                    IF (Wake_Up < 6000) OR (BMS_Voltage < BMS_Voltage_Min) THEN 
                        (* Transition: '<S1>:358' *)
                        (* Transition: '<S1>:814' *)
                        (* Exit Internal 'POWER_MOTOR_ON': '<S1>:137' *)
                        is_POWER_MOTOR_ON := UPMRacing_14E_StateMachine_IN_NO_ACTIVE_CHILD;
                        is_CAR := UPMRacing_14E_StateMachine_IN_IDLE;
                        (* Entry 'IDLE': '<S1>:333' *)
                        (* '<S1>:333:3' Cooling_Enable = false; *)
                        Cooling_Enable := FALSE;
                        (* '<S1>:333:4' [AMK_TargetVelocity1, AMK_TargetVelocity2, AMK_TargetVelocity3, AMK_TargetVelocity4... *)
                        (* '<S1>:333:5'      ]=Constant(int16(0)); *)
                        (* Simulink Function 'Constant': '<S1>:190' *)
                        x := 0;
                        i0_b_Constant(ssMethodType := SS_OUTPUT, x := x);
                        temp12 := i0_b_Constant.y1;
                        temp13 := i0_b_Constant.y2;
                        temp14 := i0_b_Constant.y3;
                        temp15 := i0_b_Constant.y4;
                        OutportBufferFory4 := temp15;
                        OutportBufferFory3 := temp14;
                        OutportBufferFory2 := temp13;
                        x_l := temp12;
                        AMK_TargetVelocity1 := x_l;
                        AMK_TargetVelocity2 := OutportBufferFory2;
                        AMK_TargetVelocity3 := OutportBufferFory3;
                        AMK_TargetVelocity4 := OutportBufferFory4;
                        (* '<S1>:333:6' [AMK_TorqueLimitPositiv1, AMK_TorqueLimitPositiv2, AMK_TorqueLimitPositiv3,... *)
                        (* '<S1>:333:7'      AMK_TorqueLimitPositiv4]=Constant(int16(0)); *)
                        (* Simulink Function 'Constant': '<S1>:190' *)
                        x := 0;
                        i0_b_Constant(ssMethodType := SS_OUTPUT, x := x);
                        temp12 := i0_b_Constant.y1;
                        temp13 := i0_b_Constant.y2;
                        temp14 := i0_b_Constant.y3;
                        temp15 := i0_b_Constant.y4;
                        OutportBufferFory4 := temp15;
                        OutportBufferFory3 := temp14;
                        OutportBufferFory2 := temp13;
                        x_l := temp12;
                        AMK_TorqueLimitPositiv1 := x_l;
                        AMK_TorqueLimitPositiv2 := OutportBufferFory2;
                        AMK_TorqueLimitPositiv3 := OutportBufferFory3;
                        AMK_TorqueLimitPositiv4 := OutportBufferFory4;
                        (* '<S1>:333:8' [AMK_TorqueLimitNegativ1, AMK_TorqueLimitNegativ2, AMK_TorqueLimitNegativ3, ... *)
                        (* '<S1>:333:9'      AMK_TorqueLimitNegativ4]=Constant(int16(0)); *)
                        (* Simulink Function 'Constant': '<S1>:190' *)
                        x := 0;
                        i0_b_Constant(ssMethodType := SS_OUTPUT, x := x);
                        temp12 := i0_b_Constant.y1;
                        temp13 := i0_b_Constant.y2;
                        temp14 := i0_b_Constant.y3;
                        temp15 := i0_b_Constant.y4;
                        OutportBufferFory4 := temp15;
                        OutportBufferFory3 := temp14;
                        OutportBufferFory2 := temp13;
                        x_l := temp12;
                        AMK_TorqueLimitNegativ1 := x_l;
                        AMK_TorqueLimitNegativ2 := OutportBufferFory2;
                        AMK_TorqueLimitNegativ3 := OutportBufferFory3;
                        AMK_TorqueLimitNegativ4 := OutportBufferFory4;
                        (* Entry Internal 'IDLE': '<S1>:333' *)
                        (* Transition: '<S1>:335' *)
                        is_IDLE := UPMRacing_14E_StateMachine_IN_LVMS_ON;
                        (* Entry 'LVMS_ON': '<S1>:334' *)
                        (* In this state the ECU is waiting to start the inizialization of the inverters *)
                        (* Right now all LV systems are starting to initialize *)
                        (* '<S1>:334:4' Estado = 1; *)
                        Estado := 1;
                        (* Battery relays *)
                        (* '<S1>:334:6' Pre_Charge = false; *)
                        Pre_Charge := FALSE;
                        (* Inverters shutdown *)
                        (* '<S1>:334:8' AMK_bInverterOn1=false; *)
                        AMK_bInverterOn1 := FALSE;
                        (* '<S1>:334:9' AMK_bInverterOn2=false; *)
                        AMK_bInverterOn2 := FALSE;
                        (* '<S1>:334:10' AMK_bInverterOn3=false; *)
                        AMK_bInverterOn3 := FALSE;
                        (* '<S1>:334:11' AMK_bInverterOn4=false; *)
                        AMK_bInverterOn4 := FALSE;
                        (* '<S1>:334:12' AMK_bEnable1=false; *)
                        AMK_bEnable1 := FALSE;
                        (* '<S1>:334:13' AMK_bEnable2=false; *)
                        AMK_bEnable2 := FALSE;
                        (* '<S1>:334:14' AMK_bEnable3=false; *)
                        AMK_bEnable3 := FALSE;
                        (* '<S1>:334:15' AMK_bEnable4=false; *)
                        AMK_bEnable4 := FALSE;
                        (* '<S1>:334:16' AMK_bDcOn1=false; *)
                        AMK_bDcOn1 := FALSE;
                        (* '<S1>:334:17' AMK_bDcOn2=false; *)
                        AMK_bDcOn2 := FALSE;
                        (* '<S1>:334:18' AMK_bDcOn3=false; *)
                        AMK_bDcOn3 := FALSE;
                        (* '<S1>:334:19' AMK_bDcOn4=false; *)
                        AMK_bDcOn4 := FALSE;
                    ELSE 
                        (* '<S1>:814:1' sf_internal_predicateOutput = BMS_Voltage < BMS_Voltage_Min; *)
                        (* Initializes as 0 all control parameters *)
                        (* '<S1>:137:5' [AMK_TargetVelocity1, AMK_TargetVelocity2, AMK_TargetVelocity3, AMK_TargetVelocity4]=Constant(int16(0)) *)
                        (* Simulink Function 'Constant': '<S1>:190' *)
                        x := 0;
                        i0_b_Constant(ssMethodType := SS_OUTPUT, x := x);
                        temp12 := i0_b_Constant.y1;
                        temp13 := i0_b_Constant.y2;
                        temp14 := i0_b_Constant.y3;
                        temp15 := i0_b_Constant.y4;
                        OutportBufferFory4 := temp15;
                        OutportBufferFory3 := temp14;
                        OutportBufferFory2 := temp13;
                        x_l := temp12;
                        AMK_TargetVelocity1 := x_l;
                        AMK_TargetVelocity2 := OutportBufferFory2;
                        AMK_TargetVelocity3 := OutportBufferFory3;
                        AMK_TargetVelocity4 := OutportBufferFory4;
                        (* '<S1>:137:6' [AMK_TorqueLimitPositiv1, AMK_TorqueLimitPositiv2, AMK_TorqueLimitPositiv3, AMK_TorqueLimitPositiv4]=Constant(int16(0)) *)
                        (* Simulink Function 'Constant': '<S1>:190' *)
                        x := 0;
                        i0_b_Constant(ssMethodType := SS_OUTPUT, x := x);
                        temp12 := i0_b_Constant.y1;
                        temp13 := i0_b_Constant.y2;
                        temp14 := i0_b_Constant.y3;
                        temp15 := i0_b_Constant.y4;
                        OutportBufferFory4 := temp15;
                        OutportBufferFory3 := temp14;
                        OutportBufferFory2 := temp13;
                        x_l := temp12;
                        AMK_TorqueLimitPositiv1 := x_l;
                        AMK_TorqueLimitPositiv2 := OutportBufferFory2;
                        AMK_TorqueLimitPositiv3 := OutportBufferFory3;
                        AMK_TorqueLimitPositiv4 := OutportBufferFory4;
                        (* '<S1>:137:7' [AMK_TorqueLimitNegativ1, AMK_TorqueLimitNegativ2, AMK_TorqueLimitNegativ3, AMK_TorqueLimitNegativ4]=Constant(int16(0)) *)
                        (* Simulink Function 'Constant': '<S1>:190' *)
                        x := 0;
                        i0_b_Constant(ssMethodType := SS_OUTPUT, x := x);
                        temp12 := i0_b_Constant.y1;
                        temp13 := i0_b_Constant.y2;
                        temp14 := i0_b_Constant.y3;
                        temp15 := i0_b_Constant.y4;
                        OutportBufferFory4 := temp15;
                        OutportBufferFory3 := temp14;
                        OutportBufferFory2 := temp13;
                        x_l := temp12;
                        AMK_TorqueLimitNegativ1 := x_l;
                        AMK_TorqueLimitNegativ2 := OutportBufferFory2;
                        AMK_TorqueLimitNegativ3 := OutportBufferFory3;
                        AMK_TorqueLimitNegativ4 := OutportBufferFory4;

                        CASE is_POWER_MOTOR_ON OF
                            UPMRacing_14E_StateMachine_IN_HV_STARTUP_1: 
                                (* During 'HV_STARTUP_1': '<S1>:144' *)
                                (* '<S1>:364:1' sf_internal_predicateOutput = AMK_bDcOn1_check==true &amp; AMK_bDcOn2_check==true &amp; AMK_bDcOn3_check==true &amp; AMK_bDcOn4_check==true; *)

                                IF ((AMK_bDcOn1_check AND AMK_bDcOn2_check) AND AMK_bDcOn3_check) AND AMK_bDcOn4_check THEN 
                                    (* Transition: '<S1>:364' *)
                                    is_POWER_MOTOR_ON := UPMRacing_14E_StateMachine_IN_INIT_PRECHARGE;
                                    temporalCounter_i1(timerAction := 1, maxTime := 0);
                                    (* Entry 'INIT_PRECHARGE': '<S1>:440' *)
                                    (* Senal que de inicio a la precarga. En el caso en que volvamos de un error, al detectar directamente *)
                                    (* que se cumple la condicion de salida, no volvera a mandar la senal de iniciar precarga. *)
                                    (* '<S1>:440:4' Estado = 13; *)
                                    Estado := 13;
                                END_IF;

                            UPMRacing_14E_StateMachine_IN_HV_STARTUP_2: 
                                (* During 'HV_STARTUP_2': '<S1>:363' *)
                                (* '<S1>:365:1' sf_internal_predicateOutput = AMK_bEnable1==true &amp; AMK_bEnable2==true &amp; AMK_bEnable3==true &amp; AMK_bEnable4==true; *)

                                IF ((AMK_bEnable1 AND AMK_bEnable2) AND AMK_bEnable3) AND AMK_bEnable4 THEN 
                                    (* Transition: '<S1>:365' *)
                                    is_POWER_MOTOR_ON := UPMRacing_14E_StateMachine_IN_HV_STARTUP_3;
                                    (* Entry 'HV_STARTUP_3': '<S1>:362' *)
                                    (* '<S1>:362:3' AMK_bEnable1=false; *)
                                    AMK_bEnable1 := FALSE;
                                    (* '<S1>:362:4' AMK_bEnable2=false; *)
                                    AMK_bEnable2 := FALSE;
                                    (* '<S1>:362:5' AMK_bEnable3=false; *)
                                    AMK_bEnable3 := FALSE;
                                    (* '<S1>:362:6' AMK_bEnable4=false; *)
                                    AMK_bEnable4 := FALSE;
                                    (* '<S1>:362:7' Estado = 15; *)
                                    Estado := 15;
                                ELSE 
                                    (* Transition: '<S1>:628' *)
                                    (* Transition: '<S1>:627' *)
                                    (* '<S1>:616:1' sf_internal_predicateOutput = Shutdown_Circuit<6000; *)

                                    IF Shutdown_Circuit < 6000 THEN 
                                        (* Transition: '<S1>:616' *)
                                        is_POWER_MOTOR_ON := UPMRacing_14E_StateMachine_IN_NO_ACTIVE_CHILD;
                                        is_CAR := UPMRacing_14E_StateMachine_IN_IDLE;
                                        (* Entry 'IDLE': '<S1>:333' *)
                                        (* '<S1>:333:3' Cooling_Enable = false; *)
                                        Cooling_Enable := FALSE;
                                        (* '<S1>:333:4' [AMK_TargetVelocity1, AMK_TargetVelocity2, AMK_TargetVelocity3, AMK_TargetVelocity4... *)
                                        (* '<S1>:333:5'      ]=Constant(int16(0)); *)
                                        (* Simulink Function 'Constant': '<S1>:190' *)
                                        x := 0;
                                        i0_b_Constant(ssMethodType := SS_OUTPUT, x := x);
                                        temp12 := i0_b_Constant.y1;
                                        temp13 := i0_b_Constant.y2;
                                        temp14 := i0_b_Constant.y3;
                                        temp15 := i0_b_Constant.y4;
                                        OutportBufferFory4 := temp15;
                                        OutportBufferFory3 := temp14;
                                        OutportBufferFory2 := temp13;
                                        x_l := temp12;
                                        AMK_TargetVelocity1 := x_l;
                                        AMK_TargetVelocity2 := OutportBufferFory2;
                                        AMK_TargetVelocity3 := OutportBufferFory3;
                                        AMK_TargetVelocity4 := OutportBufferFory4;
                                        (* '<S1>:333:6' [AMK_TorqueLimitPositiv1, AMK_TorqueLimitPositiv2, AMK_TorqueLimitPositiv3,... *)
                                        (* '<S1>:333:7'      AMK_TorqueLimitPositiv4]=Constant(int16(0)); *)
                                        (* Simulink Function 'Constant': '<S1>:190' *)
                                        x := 0;
                                        i0_b_Constant(ssMethodType := SS_OUTPUT, x := x);
                                        temp12 := i0_b_Constant.y1;
                                        temp13 := i0_b_Constant.y2;
                                        temp14 := i0_b_Constant.y3;
                                        temp15 := i0_b_Constant.y4;
                                        OutportBufferFory4 := temp15;
                                        OutportBufferFory3 := temp14;
                                        OutportBufferFory2 := temp13;
                                        x_l := temp12;
                                        AMK_TorqueLimitPositiv1 := x_l;
                                        AMK_TorqueLimitPositiv2 := OutportBufferFory2;
                                        AMK_TorqueLimitPositiv3 := OutportBufferFory3;
                                        AMK_TorqueLimitPositiv4 := OutportBufferFory4;
                                        (* '<S1>:333:8' [AMK_TorqueLimitNegativ1, AMK_TorqueLimitNegativ2, AMK_TorqueLimitNegativ3, ... *)
                                        (* '<S1>:333:9'      AMK_TorqueLimitNegativ4]=Constant(int16(0)); *)
                                        (* Simulink Function 'Constant': '<S1>:190' *)
                                        x := 0;
                                        i0_b_Constant(ssMethodType := SS_OUTPUT, x := x);
                                        temp12 := i0_b_Constant.y1;
                                        temp13 := i0_b_Constant.y2;
                                        temp14 := i0_b_Constant.y3;
                                        temp15 := i0_b_Constant.y4;
                                        OutportBufferFory4 := temp15;
                                        OutportBufferFory3 := temp14;
                                        OutportBufferFory2 := temp13;
                                        x_l := temp12;
                                        AMK_TorqueLimitNegativ1 := x_l;
                                        AMK_TorqueLimitNegativ2 := OutportBufferFory2;
                                        AMK_TorqueLimitNegativ3 := OutportBufferFory3;
                                        AMK_TorqueLimitNegativ4 := OutportBufferFory4;
                                        is_IDLE := UPMRacing_14E_StateMachine_IN_ERROR_PRECHARGE;
                                        (* Entry 'ERROR_PRECHARGE': '<S1>:617' *)
                                        (* '<S1>:617:2' Estado = 70; *)
                                        Estado := 70;
                                        (* '<S1>:617:3' Pre_Charge = false; *)
                                        Pre_Charge := FALSE;
                                    END_IF;

                                END_IF;

                            UPMRacing_14E_StateMachine_IN_HV_STARTUP_3: 
                                (* During 'HV_STARTUP_3': '<S1>:362' *)
                                (* '<S1>:208:1' sf_internal_predicateOutput = AMK_bEnable1==false &amp; AMK_bEnable2==false &amp; AMK_bEnable3==false &amp; AMK_bEnable4==false; *)

                                IF ((( NOT AMK_bEnable1) AND ( NOT AMK_bEnable2)) AND ( NOT AMK_bEnable3)) AND ( NOT AMK_bEnable4) THEN 
                                    (* Transition: '<S1>:208' *)
                                    is_POWER_MOTOR_ON := UPMRacing_14E_StateMachine_IN_HV_STARTUP_4;
                                    (* Entry 'HV_STARTUP_4': '<S1>:139' *)
                                    (* '<S1>:139:3' AMK_bEnable1=true; *)
                                    AMK_bEnable1 := TRUE;
                                    (* '<S1>:139:4' AMK_bEnable2=true; *)
                                    AMK_bEnable2 := TRUE;
                                    (* '<S1>:139:5' AMK_bEnable3=true; *)
                                    AMK_bEnable3 := TRUE;
                                    (* '<S1>:139:6' AMK_bEnable4=true; *)
                                    AMK_bEnable4 := TRUE;
                                    (* '<S1>:139:7' Estado = 16; *)
                                    Estado := 16;
                                ELSE 
                                    (* Transition: '<S1>:629' *)
                                    (* Transition: '<S1>:626' *)
                                    (* Transition: '<S1>:627' *)
                                    (* '<S1>:616:1' sf_internal_predicateOutput = Shutdown_Circuit<6000; *)

                                    IF Shutdown_Circuit < 6000 THEN 
                                        (* Transition: '<S1>:616' *)
                                        is_POWER_MOTOR_ON := UPMRacing_14E_StateMachine_IN_NO_ACTIVE_CHILD;
                                        is_CAR := UPMRacing_14E_StateMachine_IN_IDLE;
                                        (* Entry 'IDLE': '<S1>:333' *)
                                        (* '<S1>:333:3' Cooling_Enable = false; *)
                                        Cooling_Enable := FALSE;
                                        (* '<S1>:333:4' [AMK_TargetVelocity1, AMK_TargetVelocity2, AMK_TargetVelocity3, AMK_TargetVelocity4... *)
                                        (* '<S1>:333:5'      ]=Constant(int16(0)); *)
                                        (* Simulink Function 'Constant': '<S1>:190' *)
                                        x := 0;
                                        i0_b_Constant(ssMethodType := SS_OUTPUT, x := x);
                                        temp12 := i0_b_Constant.y1;
                                        temp13 := i0_b_Constant.y2;
                                        temp14 := i0_b_Constant.y3;
                                        temp15 := i0_b_Constant.y4;
                                        OutportBufferFory4 := temp15;
                                        OutportBufferFory3 := temp14;
                                        OutportBufferFory2 := temp13;
                                        x_l := temp12;
                                        AMK_TargetVelocity1 := x_l;
                                        AMK_TargetVelocity2 := OutportBufferFory2;
                                        AMK_TargetVelocity3 := OutportBufferFory3;
                                        AMK_TargetVelocity4 := OutportBufferFory4;
                                        (* '<S1>:333:6' [AMK_TorqueLimitPositiv1, AMK_TorqueLimitPositiv2, AMK_TorqueLimitPositiv3,... *)
                                        (* '<S1>:333:7'      AMK_TorqueLimitPositiv4]=Constant(int16(0)); *)
                                        (* Simulink Function 'Constant': '<S1>:190' *)
                                        x := 0;
                                        i0_b_Constant(ssMethodType := SS_OUTPUT, x := x);
                                        temp12 := i0_b_Constant.y1;
                                        temp13 := i0_b_Constant.y2;
                                        temp14 := i0_b_Constant.y3;
                                        temp15 := i0_b_Constant.y4;
                                        OutportBufferFory4 := temp15;
                                        OutportBufferFory3 := temp14;
                                        OutportBufferFory2 := temp13;
                                        x_l := temp12;
                                        AMK_TorqueLimitPositiv1 := x_l;
                                        AMK_TorqueLimitPositiv2 := OutportBufferFory2;
                                        AMK_TorqueLimitPositiv3 := OutportBufferFory3;
                                        AMK_TorqueLimitPositiv4 := OutportBufferFory4;
                                        (* '<S1>:333:8' [AMK_TorqueLimitNegativ1, AMK_TorqueLimitNegativ2, AMK_TorqueLimitNegativ3, ... *)
                                        (* '<S1>:333:9'      AMK_TorqueLimitNegativ4]=Constant(int16(0)); *)
                                        (* Simulink Function 'Constant': '<S1>:190' *)
                                        x := 0;
                                        i0_b_Constant(ssMethodType := SS_OUTPUT, x := x);
                                        temp12 := i0_b_Constant.y1;
                                        temp13 := i0_b_Constant.y2;
                                        temp14 := i0_b_Constant.y3;
                                        temp15 := i0_b_Constant.y4;
                                        OutportBufferFory4 := temp15;
                                        OutportBufferFory3 := temp14;
                                        OutportBufferFory2 := temp13;
                                        x_l := temp12;
                                        AMK_TorqueLimitNegativ1 := x_l;
                                        AMK_TorqueLimitNegativ2 := OutportBufferFory2;
                                        AMK_TorqueLimitNegativ3 := OutportBufferFory3;
                                        AMK_TorqueLimitNegativ4 := OutportBufferFory4;
                                        is_IDLE := UPMRacing_14E_StateMachine_IN_ERROR_PRECHARGE;
                                        (* Entry 'ERROR_PRECHARGE': '<S1>:617' *)
                                        (* '<S1>:617:2' Estado = 70; *)
                                        Estado := 70;
                                        (* '<S1>:617:3' Pre_Charge = false; *)
                                        Pre_Charge := FALSE;
                                    END_IF;

                                END_IF;

                            UPMRacing_14E_StateMachine_IN_HV_STARTUP_4: 
                                (* During 'HV_STARTUP_4': '<S1>:139' *)
                                (* '<S1>:367:1' sf_internal_predicateOutput = AMK_bEnable1==true &amp;  AMK_bEnable2==true &amp; ... *)
                                (* '<S1>:367:2'  AMK_bEnable3==true &amp; AMK_bEnable4==true; *)

                                IF ((AMK_bEnable1 AND AMK_bEnable2) AND AMK_bEnable3) AND AMK_bEnable4 THEN 
                                    (* Transition: '<S1>:367' *)
                                    is_POWER_MOTOR_ON := UPMRacing_14E_StateMachine_IN_HV_STARTUP_5;
                                    (* Entry 'HV_STARTUP_5': '<S1>:366' *)
                                    (* '<S1>:366:3' AMK_bInverterOn1=true; *)
                                    AMK_bInverterOn1 := TRUE;
                                    (* '<S1>:366:4' AMK_bInverterOn2=true; *)
                                    AMK_bInverterOn2 := TRUE;
                                    (* '<S1>:366:5' AMK_bInverterOn3=true; *)
                                    AMK_bInverterOn3 := TRUE;
                                    (* '<S1>:366:6' AMK_bInverterOn4=true; *)
                                    AMK_bInverterOn4 := TRUE;
                                    (* '<S1>:366:7' Estado = 17; *)
                                    Estado := 17;
                                ELSE 
                                    (* Transition: '<S1>:630' *)
                                    (* Transition: '<S1>:625' *)
                                    (* Transition: '<S1>:626' *)
                                    (* Transition: '<S1>:627' *)
                                    (* '<S1>:616:1' sf_internal_predicateOutput = Shutdown_Circuit<6000; *)

                                    IF Shutdown_Circuit < 6000 THEN 
                                        (* Transition: '<S1>:616' *)
                                        is_POWER_MOTOR_ON := UPMRacing_14E_StateMachine_IN_NO_ACTIVE_CHILD;
                                        is_CAR := UPMRacing_14E_StateMachine_IN_IDLE;
                                        (* Entry 'IDLE': '<S1>:333' *)
                                        (* '<S1>:333:3' Cooling_Enable = false; *)
                                        Cooling_Enable := FALSE;
                                        (* '<S1>:333:4' [AMK_TargetVelocity1, AMK_TargetVelocity2, AMK_TargetVelocity3, AMK_TargetVelocity4... *)
                                        (* '<S1>:333:5'      ]=Constant(int16(0)); *)
                                        (* Simulink Function 'Constant': '<S1>:190' *)
                                        x := 0;
                                        i0_b_Constant(ssMethodType := SS_OUTPUT, x := x);
                                        temp12 := i0_b_Constant.y1;
                                        temp13 := i0_b_Constant.y2;
                                        temp14 := i0_b_Constant.y3;
                                        temp15 := i0_b_Constant.y4;
                                        OutportBufferFory4 := temp15;
                                        OutportBufferFory3 := temp14;
                                        OutportBufferFory2 := temp13;
                                        x_l := temp12;
                                        AMK_TargetVelocity1 := x_l;
                                        AMK_TargetVelocity2 := OutportBufferFory2;
                                        AMK_TargetVelocity3 := OutportBufferFory3;
                                        AMK_TargetVelocity4 := OutportBufferFory4;
                                        (* '<S1>:333:6' [AMK_TorqueLimitPositiv1, AMK_TorqueLimitPositiv2, AMK_TorqueLimitPositiv3,... *)
                                        (* '<S1>:333:7'      AMK_TorqueLimitPositiv4]=Constant(int16(0)); *)
                                        (* Simulink Function 'Constant': '<S1>:190' *)
                                        x := 0;
                                        i0_b_Constant(ssMethodType := SS_OUTPUT, x := x);
                                        temp12 := i0_b_Constant.y1;
                                        temp13 := i0_b_Constant.y2;
                                        temp14 := i0_b_Constant.y3;
                                        temp15 := i0_b_Constant.y4;
                                        OutportBufferFory4 := temp15;
                                        OutportBufferFory3 := temp14;
                                        OutportBufferFory2 := temp13;
                                        x_l := temp12;
                                        AMK_TorqueLimitPositiv1 := x_l;
                                        AMK_TorqueLimitPositiv2 := OutportBufferFory2;
                                        AMK_TorqueLimitPositiv3 := OutportBufferFory3;
                                        AMK_TorqueLimitPositiv4 := OutportBufferFory4;
                                        (* '<S1>:333:8' [AMK_TorqueLimitNegativ1, AMK_TorqueLimitNegativ2, AMK_TorqueLimitNegativ3, ... *)
                                        (* '<S1>:333:9'      AMK_TorqueLimitNegativ4]=Constant(int16(0)); *)
                                        (* Simulink Function 'Constant': '<S1>:190' *)
                                        x := 0;
                                        i0_b_Constant(ssMethodType := SS_OUTPUT, x := x);
                                        temp12 := i0_b_Constant.y1;
                                        temp13 := i0_b_Constant.y2;
                                        temp14 := i0_b_Constant.y3;
                                        temp15 := i0_b_Constant.y4;
                                        OutportBufferFory4 := temp15;
                                        OutportBufferFory3 := temp14;
                                        OutportBufferFory2 := temp13;
                                        x_l := temp12;
                                        AMK_TorqueLimitNegativ1 := x_l;
                                        AMK_TorqueLimitNegativ2 := OutportBufferFory2;
                                        AMK_TorqueLimitNegativ3 := OutportBufferFory3;
                                        AMK_TorqueLimitNegativ4 := OutportBufferFory4;
                                        is_IDLE := UPMRacing_14E_StateMachine_IN_ERROR_PRECHARGE;
                                        (* Entry 'ERROR_PRECHARGE': '<S1>:617' *)
                                        (* '<S1>:617:2' Estado = 70; *)
                                        Estado := 70;
                                        (* '<S1>:617:3' Pre_Charge = false; *)
                                        Pre_Charge := FALSE;
                                    END_IF;

                                END_IF;

                            UPMRacing_14E_StateMachine_IN_HV_STARTUP_5: 
                                (* During 'HV_STARTUP_5': '<S1>:366' *)
                                (* '<S1>:262:1' sf_internal_predicateOutput = AMK_bInverterOn1_check==true &amp;  AMK_bInverterOn2_check==true &amp; ... *)
                                (* '<S1>:262:2'  AMK_bInverterOn3_check==true &amp; AMK_bInverterOn4_check==true; *)

                                IF ((AMK_bInverterOn1_check AND AMK_bInverterOn2_check) AND AMK_bInverterOn3_check) AND AMK_bInverterOn4_check THEN 
                                    (* Transition: '<S1>:262' *)
                                    is_POWER_MOTOR_ON := UPMRacing_14E_StateMachine_IN_HV_STARTUP_6;
                                    (* Entry 'HV_STARTUP_6': '<S1>:259' *)
                                    (* AMK_X140_BE2_INV_1=true; *)
                                    (* AMK_X140_BE2_INV_2=true; *)
                                    (* AMK_X140_BE2_INV_3=true; *)
                                    (* AMK_X140_BE2_INV_4=true; *)
                                    (* '<S1>:259:7' Estado = 18; *)
                                    Estado := 18;
                                ELSE 
                                    (* Transition: '<S1>:631' *)
                                    (* Transition: '<S1>:624' *)
                                    (* Transition: '<S1>:625' *)
                                    (* Transition: '<S1>:626' *)
                                    (* Transition: '<S1>:627' *)
                                    (* '<S1>:616:1' sf_internal_predicateOutput = Shutdown_Circuit<6000; *)

                                    IF Shutdown_Circuit < 6000 THEN 
                                        (* Transition: '<S1>:616' *)
                                        is_POWER_MOTOR_ON := UPMRacing_14E_StateMachine_IN_NO_ACTIVE_CHILD;
                                        is_CAR := UPMRacing_14E_StateMachine_IN_IDLE;
                                        (* Entry 'IDLE': '<S1>:333' *)
                                        (* '<S1>:333:3' Cooling_Enable = false; *)
                                        Cooling_Enable := FALSE;
                                        (* '<S1>:333:4' [AMK_TargetVelocity1, AMK_TargetVelocity2, AMK_TargetVelocity3, AMK_TargetVelocity4... *)
                                        (* '<S1>:333:5'      ]=Constant(int16(0)); *)
                                        (* Simulink Function 'Constant': '<S1>:190' *)
                                        x := 0;
                                        i0_b_Constant(ssMethodType := SS_OUTPUT, x := x);
                                        temp12 := i0_b_Constant.y1;
                                        temp13 := i0_b_Constant.y2;
                                        temp14 := i0_b_Constant.y3;
                                        temp15 := i0_b_Constant.y4;
                                        OutportBufferFory4 := temp15;
                                        OutportBufferFory3 := temp14;
                                        OutportBufferFory2 := temp13;
                                        x_l := temp12;
                                        AMK_TargetVelocity1 := x_l;
                                        AMK_TargetVelocity2 := OutportBufferFory2;
                                        AMK_TargetVelocity3 := OutportBufferFory3;
                                        AMK_TargetVelocity4 := OutportBufferFory4;
                                        (* '<S1>:333:6' [AMK_TorqueLimitPositiv1, AMK_TorqueLimitPositiv2, AMK_TorqueLimitPositiv3,... *)
                                        (* '<S1>:333:7'      AMK_TorqueLimitPositiv4]=Constant(int16(0)); *)
                                        (* Simulink Function 'Constant': '<S1>:190' *)
                                        x := 0;
                                        i0_b_Constant(ssMethodType := SS_OUTPUT, x := x);
                                        temp12 := i0_b_Constant.y1;
                                        temp13 := i0_b_Constant.y2;
                                        temp14 := i0_b_Constant.y3;
                                        temp15 := i0_b_Constant.y4;
                                        OutportBufferFory4 := temp15;
                                        OutportBufferFory3 := temp14;
                                        OutportBufferFory2 := temp13;
                                        x_l := temp12;
                                        AMK_TorqueLimitPositiv1 := x_l;
                                        AMK_TorqueLimitPositiv2 := OutportBufferFory2;
                                        AMK_TorqueLimitPositiv3 := OutportBufferFory3;
                                        AMK_TorqueLimitPositiv4 := OutportBufferFory4;
                                        (* '<S1>:333:8' [AMK_TorqueLimitNegativ1, AMK_TorqueLimitNegativ2, AMK_TorqueLimitNegativ3, ... *)
                                        (* '<S1>:333:9'      AMK_TorqueLimitNegativ4]=Constant(int16(0)); *)
                                        (* Simulink Function 'Constant': '<S1>:190' *)
                                        x := 0;
                                        i0_b_Constant(ssMethodType := SS_OUTPUT, x := x);
                                        temp12 := i0_b_Constant.y1;
                                        temp13 := i0_b_Constant.y2;
                                        temp14 := i0_b_Constant.y3;
                                        temp15 := i0_b_Constant.y4;
                                        OutportBufferFory4 := temp15;
                                        OutportBufferFory3 := temp14;
                                        OutportBufferFory2 := temp13;
                                        x_l := temp12;
                                        AMK_TorqueLimitNegativ1 := x_l;
                                        AMK_TorqueLimitNegativ2 := OutportBufferFory2;
                                        AMK_TorqueLimitNegativ3 := OutportBufferFory3;
                                        AMK_TorqueLimitNegativ4 := OutportBufferFory4;
                                        is_IDLE := UPMRacing_14E_StateMachine_IN_ERROR_PRECHARGE;
                                        (* Entry 'ERROR_PRECHARGE': '<S1>:617' *)
                                        (* '<S1>:617:2' Estado = 70; *)
                                        Estado := 70;
                                        (* '<S1>:617:3' Pre_Charge = false; *)
                                        Pre_Charge := FALSE;
                                    END_IF;

                                END_IF;

                            UPMRacing_14E_StateMachine_IN_HV_STARTUP_6: 
                                (* During 'HV_STARTUP_6': '<S1>:259' *)
                                (* '<S1>:147:1' sf_internal_predicateOutput = AMK_bQuitInverterOn1==true &amp;  AMK_bQuitInverterOn2==true... *)
                                (* '<S1>:147:2'  &amp; AMK_bQuitInverterOn3==true &amp; AMK_bQuitInverterOn4==true... *)
                                (* '<S1>:147:3' &amp; Drive_Button < 12000; *)

                                IF (((AMK_bQuitInverterOn1 AND AMK_bQuitInverterOn2) AND AMK_bQuitInverterOn3) AND AMK_bQuitInverterOn4) AND (Drive_Button < 12000) THEN 
                                    (* Transition: '<S1>:147' *)
                                    is_POWER_MOTOR_ON := UPMRacing_14E_StateMachine_IN_NO_ACTIVE_CHILD;
                                    is_CAR := UPMRacing_14E_StateMachine_IN_DRIVE;
                                    (* Entry 'DRIVE': '<S1>:169' *)
                                    (* '<S1>:169:2' Cooling_Enable = true; *)
                                    Cooling_Enable := TRUE;
                                    (* Entry Internal 'DRIVE': '<S1>:169' *)
                                    (* Transition: '<S1>:264' *)
                                    is_DRIVE := UPMRacing_14E_StateMachine_IN_PRE_DRIVE;
                                    (* Entry 'PRE_DRIVE': '<S1>:503' *)
                                    (* '<S1>:503:2' Estado = 20; *)
                                    Estado := 20;
                                ELSE 
                                    (* Transition: '<S1>:634' *)
                                    (* Transition: '<S1>:633' *)
                                    (* Transition: '<S1>:624' *)
                                    (* Transition: '<S1>:625' *)
                                    (* Transition: '<S1>:626' *)
                                    (* Transition: '<S1>:627' *)
                                    (* '<S1>:616:1' sf_internal_predicateOutput = Shutdown_Circuit<6000; *)

                                    IF Shutdown_Circuit < 6000 THEN 
                                        (* Transition: '<S1>:616' *)
                                        is_POWER_MOTOR_ON := UPMRacing_14E_StateMachine_IN_NO_ACTIVE_CHILD;
                                        is_CAR := UPMRacing_14E_StateMachine_IN_IDLE;
                                        (* Entry 'IDLE': '<S1>:333' *)
                                        (* '<S1>:333:3' Cooling_Enable = false; *)
                                        Cooling_Enable := FALSE;
                                        (* '<S1>:333:4' [AMK_TargetVelocity1, AMK_TargetVelocity2, AMK_TargetVelocity3, AMK_TargetVelocity4... *)
                                        (* '<S1>:333:5'      ]=Constant(int16(0)); *)
                                        (* Simulink Function 'Constant': '<S1>:190' *)
                                        x := 0;
                                        i0_b_Constant(ssMethodType := SS_OUTPUT, x := x);
                                        temp12 := i0_b_Constant.y1;
                                        temp13 := i0_b_Constant.y2;
                                        temp14 := i0_b_Constant.y3;
                                        temp15 := i0_b_Constant.y4;
                                        OutportBufferFory4 := temp15;
                                        OutportBufferFory3 := temp14;
                                        OutportBufferFory2 := temp13;
                                        x_l := temp12;
                                        AMK_TargetVelocity1 := x_l;
                                        AMK_TargetVelocity2 := OutportBufferFory2;
                                        AMK_TargetVelocity3 := OutportBufferFory3;
                                        AMK_TargetVelocity4 := OutportBufferFory4;
                                        (* '<S1>:333:6' [AMK_TorqueLimitPositiv1, AMK_TorqueLimitPositiv2, AMK_TorqueLimitPositiv3,... *)
                                        (* '<S1>:333:7'      AMK_TorqueLimitPositiv4]=Constant(int16(0)); *)
                                        (* Simulink Function 'Constant': '<S1>:190' *)
                                        x := 0;
                                        i0_b_Constant(ssMethodType := SS_OUTPUT, x := x);
                                        temp12 := i0_b_Constant.y1;
                                        temp13 := i0_b_Constant.y2;
                                        temp14 := i0_b_Constant.y3;
                                        temp15 := i0_b_Constant.y4;
                                        OutportBufferFory4 := temp15;
                                        OutportBufferFory3 := temp14;
                                        OutportBufferFory2 := temp13;
                                        x_l := temp12;
                                        AMK_TorqueLimitPositiv1 := x_l;
                                        AMK_TorqueLimitPositiv2 := OutportBufferFory2;
                                        AMK_TorqueLimitPositiv3 := OutportBufferFory3;
                                        AMK_TorqueLimitPositiv4 := OutportBufferFory4;
                                        (* '<S1>:333:8' [AMK_TorqueLimitNegativ1, AMK_TorqueLimitNegativ2, AMK_TorqueLimitNegativ3, ... *)
                                        (* '<S1>:333:9'      AMK_TorqueLimitNegativ4]=Constant(int16(0)); *)
                                        (* Simulink Function 'Constant': '<S1>:190' *)
                                        x := 0;
                                        i0_b_Constant(ssMethodType := SS_OUTPUT, x := x);
                                        temp12 := i0_b_Constant.y1;
                                        temp13 := i0_b_Constant.y2;
                                        temp14 := i0_b_Constant.y3;
                                        temp15 := i0_b_Constant.y4;
                                        OutportBufferFory4 := temp15;
                                        OutportBufferFory3 := temp14;
                                        OutportBufferFory2 := temp13;
                                        x_l := temp12;
                                        AMK_TorqueLimitNegativ1 := x_l;
                                        AMK_TorqueLimitNegativ2 := OutportBufferFory2;
                                        AMK_TorqueLimitNegativ3 := OutportBufferFory3;
                                        AMK_TorqueLimitNegativ4 := OutportBufferFory4;
                                        is_IDLE := UPMRacing_14E_StateMachine_IN_ERROR_PRECHARGE;
                                        (* Entry 'ERROR_PRECHARGE': '<S1>:617' *)
                                        (* '<S1>:617:2' Estado = 70; *)
                                        Estado := 70;
                                        (* '<S1>:617:3' Pre_Charge = false; *)
                                        Pre_Charge := FALSE;
                                    END_IF;

                                END_IF;

                            UPMRacing_14E_StateMachine_IN_INIT_PRECHARGE: 
                                (* During 'INIT_PRECHARGE': '<S1>:440' *)
                                (* '<S1>:441:1' sf_internal_predicateOutput = AMK_bQuitDcOn1==true &amp; AMK_bQuitDcOn2==true &amp; AMK_bQuitDcOn3==true &amp; AMK_bQuitDcOn4==true; *)

                                IF ((AMK_bQuitDcOn1 AND AMK_bQuitDcOn2) AND AMK_bQuitDcOn3) AND AMK_bQuitDcOn4 THEN 
                                    (* Transition: '<S1>:441' *)
                                    is_POWER_MOTOR_ON := UPMRacing_14E_StateMachine_IN_HV_STARTUP_2;
                                    (* Entry 'HV_STARTUP_2': '<S1>:363' *)
                                    (* '<S1>:363:3' AMK_bEnable1=true; *)
                                    AMK_bEnable1 := TRUE;
                                    (* '<S1>:363:4' AMK_bEnable2=true; *)
                                    AMK_bEnable2 := TRUE;
                                    (* '<S1>:363:5' AMK_bEnable3=true; *)
                                    AMK_bEnable3 := TRUE;
                                    (* '<S1>:363:6' AMK_bEnable4=true; *)
                                    AMK_bEnable4 := TRUE;
                                    (* '<S1>:363:7' Estado = 14; *)
                                    Estado := 14;
                                ELSE 
                                    (* '<S1>:615:1' sf_internal_predicateOutput = after(2,sec); *)
                                    temporalCounter_i1(timerAction := 2, maxTime := 2000);

                                    IF temporalCounter_i1.done THEN 
                                        (* Transition: '<S1>:615' *)
                                        (* '<S1>:616:1' sf_internal_predicateOutput = Shutdown_Circuit<6000; *)

                                        IF Shutdown_Circuit < 6000 THEN 
                                            (* Transition: '<S1>:616' *)
                                            is_POWER_MOTOR_ON := UPMRacing_14E_StateMachine_IN_NO_ACTIVE_CHILD;
                                            is_CAR := UPMRacing_14E_StateMachine_IN_IDLE;
                                            (* Entry 'IDLE': '<S1>:333' *)
                                            (* '<S1>:333:3' Cooling_Enable = false; *)
                                            Cooling_Enable := FALSE;
                                            (* '<S1>:333:4' [AMK_TargetVelocity1, AMK_TargetVelocity2, AMK_TargetVelocity3, AMK_TargetVelocity4... *)
                                            (* '<S1>:333:5'      ]=Constant(int16(0)); *)
                                            (* Simulink Function 'Constant': '<S1>:190' *)
                                            x := 0;
                                            i0_b_Constant(ssMethodType := SS_OUTPUT, x := x);
                                            temp12 := i0_b_Constant.y1;
                                            temp13 := i0_b_Constant.y2;
                                            temp14 := i0_b_Constant.y3;
                                            temp15 := i0_b_Constant.y4;
                                            OutportBufferFory4 := temp15;
                                            OutportBufferFory3 := temp14;
                                            OutportBufferFory2 := temp13;
                                            x_l := temp12;
                                            AMK_TargetVelocity1 := x_l;
                                            AMK_TargetVelocity2 := OutportBufferFory2;
                                            AMK_TargetVelocity3 := OutportBufferFory3;
                                            AMK_TargetVelocity4 := OutportBufferFory4;
                                            (* '<S1>:333:6' [AMK_TorqueLimitPositiv1, AMK_TorqueLimitPositiv2, AMK_TorqueLimitPositiv3,... *)
                                            (* '<S1>:333:7'      AMK_TorqueLimitPositiv4]=Constant(int16(0)); *)
                                            (* Simulink Function 'Constant': '<S1>:190' *)
                                            x := 0;
                                            i0_b_Constant(ssMethodType := SS_OUTPUT, x := x);
                                            temp12 := i0_b_Constant.y1;
                                            temp13 := i0_b_Constant.y2;
                                            temp14 := i0_b_Constant.y3;
                                            temp15 := i0_b_Constant.y4;
                                            OutportBufferFory4 := temp15;
                                            OutportBufferFory3 := temp14;
                                            OutportBufferFory2 := temp13;
                                            x_l := temp12;
                                            AMK_TorqueLimitPositiv1 := x_l;
                                            AMK_TorqueLimitPositiv2 := OutportBufferFory2;
                                            AMK_TorqueLimitPositiv3 := OutportBufferFory3;
                                            AMK_TorqueLimitPositiv4 := OutportBufferFory4;
                                            (* '<S1>:333:8' [AMK_TorqueLimitNegativ1, AMK_TorqueLimitNegativ2, AMK_TorqueLimitNegativ3, ... *)
                                            (* '<S1>:333:9'      AMK_TorqueLimitNegativ4]=Constant(int16(0)); *)
                                            (* Simulink Function 'Constant': '<S1>:190' *)
                                            x := 0;
                                            i0_b_Constant(ssMethodType := SS_OUTPUT, x := x);
                                            temp12 := i0_b_Constant.y1;
                                            temp13 := i0_b_Constant.y2;
                                            temp14 := i0_b_Constant.y3;
                                            temp15 := i0_b_Constant.y4;
                                            OutportBufferFory4 := temp15;
                                            OutportBufferFory3 := temp14;
                                            OutportBufferFory2 := temp13;
                                            x_l := temp12;
                                            AMK_TorqueLimitNegativ1 := x_l;
                                            AMK_TorqueLimitNegativ2 := OutportBufferFory2;
                                            AMK_TorqueLimitNegativ3 := OutportBufferFory3;
                                            AMK_TorqueLimitNegativ4 := OutportBufferFory4;
                                            is_IDLE := UPMRacing_14E_StateMachine_IN_ERROR_PRECHARGE;
                                            (* Entry 'ERROR_PRECHARGE': '<S1>:617' *)
                                            (* '<S1>:617:2' Estado = 70; *)
                                            Estado := 70;
                                            (* '<S1>:617:3' Pre_Charge = false; *)
                                            Pre_Charge := FALSE;
                                        ELSE 
                                            (* Senal que de inicio a la precarga. En el caso en que volvamos de un error, al detectar directamente *)
                                            (* que se cumple la condicion de salida, no volvera a mandar la senal de iniciar precarga. *)
                                            (* '<S1>:440:6' Pre_Charge=true; *)
                                            Pre_Charge := TRUE;
                                        END_IF;

                                    ELSE 
                                        (* Senal que de inicio a la precarga. En el caso en que volvamos de un error, al detectar directamente *)
                                        (* que se cumple la condicion de salida, no volvera a mandar la senal de iniciar precarga. *)
                                        (* '<S1>:440:6' Pre_Charge=true; *)
                                        Pre_Charge := TRUE;
                                    END_IF;

                                END_IF;

                            ELSE
                                (* During 'INVERTER_ON': '<S1>:163' *)
                                (* '<S1>:164:1' sf_internal_predicateOutput = AMK_bSystemReady1==true &amp; AMK_bSystemReady2==true &amp; AMK_bSystemReady3==true &amp;... *)
                                (* '<S1>:164:2' AMK_bSystemReady4==true; *)

                                IF ((AMK_bSystemReady1 AND AMK_bSystemReady2) AND AMK_bSystemReady3) AND AMK_bSystemReady4 THEN 
                                    (* Transition: '<S1>:164' *)
                                    is_POWER_MOTOR_ON := UPMRacing_14E_StateMachine_IN_HV_STARTUP_1;
                                    (* Entry 'HV_STARTUP_1': '<S1>:144' *)
                                    (* '<S1>:144:3' AMK_bDcOn1=true; *)
                                    AMK_bDcOn1 := TRUE;
                                    (* '<S1>:144:4' AMK_bDcOn2=true; *)
                                    AMK_bDcOn2 := TRUE;
                                    (* '<S1>:144:5' AMK_bDcOn3=true; *)
                                    AMK_bDcOn3 := TRUE;
                                    (* '<S1>:144:6' AMK_bDcOn4=true; *)
                                    AMK_bDcOn4 := TRUE;
                                    (* '<S1>:144:7' Estado = 12; *)
                                    Estado := 12;
                                END_IF;

                        END_CASE;

                    END_IF;

                ELSE
                    (* During 'SHUTDOWN_SEQUENCE': '<S1>:189' *)

                    CASE is_SHUTDOWN_SEQUENCE OF
                        UPMRacing_14E_StateMachine_IN_HV_SHUTDOWN: 
                            (* During 'HV_SHUTDOWN': '<S1>:216' *)
                            (* '<S1>:473:1' sf_internal_predicateOutput = AMK_bDcOn1_check==false &amp; AMK_bDcOn2_check==false &amp; AMK_bDcOn3_check==false &amp; AMK_bDcOn4_check==false; *)

                            IF ((( NOT AMK_bDcOn1_check) AND ( NOT AMK_bDcOn2_check)) AND ( NOT AMK_bDcOn3_check)) AND ( NOT AMK_bDcOn4_check) THEN 
                                (* Transition: '<S1>:473' *)
                                is_SHUTDOWN_SEQUENCE := UPMRacing_14E_StateMachine_IN_INIT_DISCHARGE;
                                temporalCounter_i1(timerAction := 1, maxTime := 0);
                                (* Entry 'INIT_DISCHARGE': '<S1>:472' *)
                                (* '<S1>:472:2' Estado = 33; *)
                                Estado := 33;
                            ELSE 
                                (* '<S1>:216:2' Estado = 32; *)
                                Estado := 32;
                                (* AMK_X140_BE1_INV_1=false; *)
                                (* AMK_X140_BE1_INV_2=false; *)
                                (* AMK_X140_BE1_INV_3=false; *)
                                (* AMK_X140_BE1_INV_4=false; *)
                                (* '<S1>:216:7' AMK_bDcOn1=false; *)
                                AMK_bDcOn1 := FALSE;
                                (* '<S1>:216:8' AMK_bDcOn2=false; *)
                                AMK_bDcOn2 := FALSE;
                                (* '<S1>:216:9' AMK_bDcOn3=false; *)
                                AMK_bDcOn3 := FALSE;
                                (* '<S1>:216:10' AMK_bDcOn4=false; *)
                                AMK_bDcOn4 := FALSE;
                            END_IF;

                        UPMRacing_14E_StateMachine_IN_INIT_DISCHARGE: 
                            (* During 'INIT_DISCHARGE': '<S1>:472' *)
                            (* '<S1>:476:1' sf_internal_predicateOutput = (Pre_Charge == false) &amp; (Shutdown_Circuit < 6000); *)

                            IF ( NOT Pre_Charge) AND (Shutdown_Circuit < 6000) THEN 
                                (* Transition: '<S1>:476' *)
                                (* '<S1>:477:1' sf_internal_predicateOutput = after(5,sec); *)
                                temporalCounter_i1(timerAction := 2, maxTime := 5000);

                                IF temporalCounter_i1.done THEN 
                                    (* Transition: '<S1>:477' *)
                                    is_SHUTDOWN_SEQUENCE := UPMRacing_14E_StateMachine_IN_INIT_DISCHARGE1;
                                    (* Entry 'INIT_DISCHARGE1': '<S1>:474' *)
                                    (* '<S1>:474:2' Estado = 34; *)
                                    Estado := 34;
                                END_IF;

                            ELSE 
                                (* '<S1>:472:4' Pre_Charge = false; *)
                                Pre_Charge := FALSE;
                            END_IF;

                        UPMRacing_14E_StateMachine_IN_INIT_DISCHARGE1: 
                            (* During 'INIT_DISCHARGE1': '<S1>:474' *)
                            (* '<S1>:221:1' sf_internal_predicateOutput = AMK_bQuitDcOn1==false &amp; AMK_bQuitDcOn2==false &amp;  AMK_bQuitDcOn3==false &amp; AMK_bQuitDcOn1==false &amp; Wake_Up < 6000; *)
                            sf_internal_predicateOutput :=  NOT AMK_bQuitDcOn1;

                            IF (((sf_internal_predicateOutput AND ( NOT AMK_bQuitDcOn2)) AND ( NOT AMK_bQuitDcOn3)) AND sf_internal_predicateOutput) AND (Wake_Up < 6000) THEN 
                                (* Transition: '<S1>:221' *)
                                is_SHUTDOWN_SEQUENCE := UPMRacing_14E_StateMachine_IN_NO_ACTIVE_CHILD;
                                is_CAR := UPMRacing_14E_StateMachine_IN_IDLE;
                                (* Entry 'IDLE': '<S1>:333' *)
                                (* '<S1>:333:3' Cooling_Enable = false; *)
                                Cooling_Enable := FALSE;
                                (* '<S1>:333:4' [AMK_TargetVelocity1, AMK_TargetVelocity2, AMK_TargetVelocity3, AMK_TargetVelocity4... *)
                                (* '<S1>:333:5'      ]=Constant(int16(0)); *)
                                (* Simulink Function 'Constant': '<S1>:190' *)
                                x := 0;
                                i0_b_Constant(ssMethodType := SS_OUTPUT, x := x);
                                temp12 := i0_b_Constant.y1;
                                temp13 := i0_b_Constant.y2;
                                temp14 := i0_b_Constant.y3;
                                temp15 := i0_b_Constant.y4;
                                OutportBufferFory4 := temp15;
                                OutportBufferFory3 := temp14;
                                OutportBufferFory2 := temp13;
                                x_l := temp12;
                                AMK_TargetVelocity1 := x_l;
                                AMK_TargetVelocity2 := OutportBufferFory2;
                                AMK_TargetVelocity3 := OutportBufferFory3;
                                AMK_TargetVelocity4 := OutportBufferFory4;
                                (* '<S1>:333:6' [AMK_TorqueLimitPositiv1, AMK_TorqueLimitPositiv2, AMK_TorqueLimitPositiv3,... *)
                                (* '<S1>:333:7'      AMK_TorqueLimitPositiv4]=Constant(int16(0)); *)
                                (* Simulink Function 'Constant': '<S1>:190' *)
                                x := 0;
                                i0_b_Constant(ssMethodType := SS_OUTPUT, x := x);
                                temp12 := i0_b_Constant.y1;
                                temp13 := i0_b_Constant.y2;
                                temp14 := i0_b_Constant.y3;
                                temp15 := i0_b_Constant.y4;
                                OutportBufferFory4 := temp15;
                                OutportBufferFory3 := temp14;
                                OutportBufferFory2 := temp13;
                                x_l := temp12;
                                AMK_TorqueLimitPositiv1 := x_l;
                                AMK_TorqueLimitPositiv2 := OutportBufferFory2;
                                AMK_TorqueLimitPositiv3 := OutportBufferFory3;
                                AMK_TorqueLimitPositiv4 := OutportBufferFory4;
                                (* '<S1>:333:8' [AMK_TorqueLimitNegativ1, AMK_TorqueLimitNegativ2, AMK_TorqueLimitNegativ3, ... *)
                                (* '<S1>:333:9'      AMK_TorqueLimitNegativ4]=Constant(int16(0)); *)
                                (* Simulink Function 'Constant': '<S1>:190' *)
                                x := 0;
                                i0_b_Constant(ssMethodType := SS_OUTPUT, x := x);
                                temp12 := i0_b_Constant.y1;
                                temp13 := i0_b_Constant.y2;
                                temp14 := i0_b_Constant.y3;
                                temp15 := i0_b_Constant.y4;
                                OutportBufferFory4 := temp15;
                                OutportBufferFory3 := temp14;
                                OutportBufferFory2 := temp13;
                                x_l := temp12;
                                AMK_TorqueLimitNegativ1 := x_l;
                                AMK_TorqueLimitNegativ2 := OutportBufferFory2;
                                AMK_TorqueLimitNegativ3 := OutportBufferFory3;
                                AMK_TorqueLimitNegativ4 := OutportBufferFory4;
                                (* Entry Internal 'IDLE': '<S1>:333' *)
                                (* Transition: '<S1>:335' *)
                                is_IDLE := UPMRacing_14E_StateMachine_IN_LVMS_ON;
                                (* Entry 'LVMS_ON': '<S1>:334' *)
                                (* In this state the ECU is waiting to start the inizialization of the inverters *)
                                (* Right now all LV systems are starting to initialize *)
                                (* '<S1>:334:4' Estado = 1; *)
                                Estado := 1;
                                (* Battery relays *)
                                (* '<S1>:334:6' Pre_Charge = false; *)
                                Pre_Charge := FALSE;
                                (* Inverters shutdown *)
                                (* '<S1>:334:8' AMK_bInverterOn1=false; *)
                                AMK_bInverterOn1 := FALSE;
                                (* '<S1>:334:9' AMK_bInverterOn2=false; *)
                                AMK_bInverterOn2 := FALSE;
                                (* '<S1>:334:10' AMK_bInverterOn3=false; *)
                                AMK_bInverterOn3 := FALSE;
                                (* '<S1>:334:11' AMK_bInverterOn4=false; *)
                                AMK_bInverterOn4 := FALSE;
                                (* '<S1>:334:12' AMK_bEnable1=false; *)
                                AMK_bEnable1 := FALSE;
                                (* '<S1>:334:13' AMK_bEnable2=false; *)
                                AMK_bEnable2 := FALSE;
                                (* '<S1>:334:14' AMK_bEnable3=false; *)
                                AMK_bEnable3 := FALSE;
                                (* '<S1>:334:15' AMK_bEnable4=false; *)
                                AMK_bEnable4 := FALSE;
                                (* '<S1>:334:16' AMK_bDcOn1=false; *)
                                AMK_bDcOn1 := FALSE;
                                (* '<S1>:334:17' AMK_bDcOn2=false; *)
                                AMK_bDcOn2 := FALSE;
                                (* '<S1>:334:18' AMK_bDcOn3=false; *)
                                AMK_bDcOn3 := FALSE;
                                (* '<S1>:334:19' AMK_bDcOn4=false; *)
                                AMK_bDcOn4 := FALSE;
                            END_IF;

                        ELSE
                            (* During 'INVERTER_CONTROLLER_SHUTDOWN': '<S1>:212' *)
                            (* '<S1>:217:1' sf_internal_predicateOutput = AMK_bQuitInverterOn1==false &amp; AMK_bQuitInverterOn2==false &amp;  AMK_bQuitInverterOn3==false &amp; AMK_bQuitInverterOn4==false... *)
                            (* '<S1>:217:2' &amp; AMK_bInverterOn1_check==false &amp;  AMK_bInverterOn2_check==false &amp;  AMK_bInverterOn3_check==false &amp; AMK_bInverterOn4_check==false; *)

                            IF ((((((( NOT AMK_bQuitInverterOn1) AND ( NOT AMK_bQuitInverterOn2)) AND ( NOT AMK_bQuitInverterOn3)) AND ( NOT AMK_bQuitInverterOn4)) AND ( NOT AMK_bInverterOn1_check)) AND ( NOT AMK_bInverterOn2_check)) AND ( NOT AMK_bInverterOn3_check)) AND ( NOT AMK_bInverterOn4_check) THEN 
                                (* Transition: '<S1>:217' *)
                                is_SHUTDOWN_SEQUENCE := UPMRacing_14E_StateMachine_IN_HV_SHUTDOWN;
                                (* Entry 'HV_SHUTDOWN': '<S1>:216' *)
                            ELSE 
                                (* '<S1>:212:2' Estado = 31; *)
                                Estado := 31;
                                (* AMK_X140_BE2_INV_1=false; *)
                                (* AMK_X140_BE2_INV_2=false; *)
                                (* AMK_X140_BE2_INV_3=false; *)
                                (* AMK_X140_BE2_INV_4=false; *)
                                (* '<S1>:212:7' AMK_bInverterOn1=false; *)
                                AMK_bInverterOn1 := FALSE;
                                (* '<S1>:212:8' AMK_bInverterOn2=false; *)
                                AMK_bInverterOn2 := FALSE;
                                (* '<S1>:212:9' AMK_bInverterOn3=false; *)
                                AMK_bInverterOn3 := FALSE;
                                (* '<S1>:212:10' AMK_bInverterOn4=false; *)
                                AMK_bInverterOn4 := FALSE;
                                (* '<S1>:212:11' AMK_bEnable1=false; *)
                                AMK_bEnable1 := FALSE;
                                (* '<S1>:212:12' AMK_bEnable2=false; *)
                                AMK_bEnable2 := FALSE;
                                (* '<S1>:212:13' AMK_bEnable3=false; *)
                                AMK_bEnable3 := FALSE;
                                (* '<S1>:212:14' AMK_bEnable4=false; *)
                                AMK_bEnable4 := FALSE;
                            END_IF;

                    END_CASE;

            END_CASE;


            IF temp9 THEN 
                (* Exit Internal 'DRIVE': '<S1>:169' *)

                CASE is_DRIVE OF
                    UPMRacing_14E_StateMachine_IN_RTDS: 
                        (* Exit 'RTDS': '<S1>:555' *)
                        (* '<S1>:555:8' RTDS_Sound = false; *)
                        RTDS_Sound := FALSE;
                        is_DRIVE := UPMRacing_14E_StateMachine_IN_NO_ACTIVE_CHILD;
                    ELSE
                        is_DRIVE := UPMRacing_14E_StateMachine_IN_NO_ACTIVE_CHILD;
                END_CASE;

                is_CAR := UPMRacing_14E_StateMachine_IN_SHUTDOWN_SEQUENCE;
                (* Entry 'SHUTDOWN_SEQUENCE': '<S1>:189' *)
                (* '<S1>:189:3' [AMK_TorqueLimitNegativ1,AMK_TorqueLimitNegativ2,AMK_TorqueLimitNegativ3,AMK_TorqueLimitNegativ4]=Constant(int16(0)); *)
                (* Simulink Function 'Constant': '<S1>:190' *)
                x := 0;
                i0_b_Constant(ssMethodType := SS_OUTPUT, x := x);
                temp12 := i0_b_Constant.y1;
                temp13 := i0_b_Constant.y2;
                temp14 := i0_b_Constant.y3;
                temp15 := i0_b_Constant.y4;
                OutportBufferFory4 := temp15;
                OutportBufferFory3 := temp14;
                OutportBufferFory2 := temp13;
                x_l := temp12;
                AMK_TorqueLimitNegativ1 := x_l;
                AMK_TorqueLimitNegativ2 := OutportBufferFory2;
                AMK_TorqueLimitNegativ3 := OutportBufferFory3;
                AMK_TorqueLimitNegativ4 := OutportBufferFory4;
                (* '<S1>:189:4' [AMK_TargetVelocity1, AMK_TargetVelocity2, AMK_TargetVelocity3,AMK_TargetVelocity4]=Constant(int16(0)); *)
                (* Simulink Function 'Constant': '<S1>:190' *)
                x := 0;
                i0_b_Constant(ssMethodType := SS_OUTPUT, x := x);
                temp12 := i0_b_Constant.y1;
                temp13 := i0_b_Constant.y2;
                temp14 := i0_b_Constant.y3;
                temp15 := i0_b_Constant.y4;
                OutportBufferFory4 := temp15;
                OutportBufferFory3 := temp14;
                OutportBufferFory2 := temp13;
                x_l := temp12;
                AMK_TargetVelocity1 := x_l;
                AMK_TargetVelocity2 := OutportBufferFory2;
                AMK_TargetVelocity3 := OutportBufferFory3;
                AMK_TargetVelocity4 := OutportBufferFory4;
                (* '<S1>:189:5' [AMK_TorqueLimitPositiv1, AMK_TorqueLimitPositiv2, AMK_TorqueLimitPositiv3,AMK_TorqueLimitPositiv4]=Constant(int16(0)); *)
                (* Simulink Function 'Constant': '<S1>:190' *)
                x := 0;
                i0_b_Constant(ssMethodType := SS_OUTPUT, x := x);
                temp12 := i0_b_Constant.y1;
                temp13 := i0_b_Constant.y2;
                temp14 := i0_b_Constant.y3;
                temp15 := i0_b_Constant.y4;
                OutportBufferFory4 := temp15;
                OutportBufferFory3 := temp14;
                OutportBufferFory2 := temp13;
                x_l := temp12;
                AMK_TorqueLimitPositiv1 := x_l;
                AMK_TorqueLimitPositiv2 := OutportBufferFory2;
                AMK_TorqueLimitPositiv3 := OutportBufferFory3;
                AMK_TorqueLimitPositiv4 := OutportBufferFory4;
                (* '<S1>:189:6' Cooling_Enable = true; *)
                Cooling_Enable := TRUE;
                (* Entry Internal 'SHUTDOWN_SEQUENCE': '<S1>:189' *)
                (* Transition: '<S1>:345' *)
                is_SHUTDOWN_SEQUENCE := UPMRacing_14E_StateMachine_IN_INVERTER_CONTROLLER_SHUTDOWN;
                (* Entry 'INVERTER_CONTROLLER_SHUTDOWN': '<S1>:212' *)
            END_IF;


            IF temp8 THEN 
                is_DRIVE := UPMRacing_14E_StateMachine_IN_BRAKE;
                (* Entry 'BRAKE': '<S1>:170' *)
                (* '<S1>:170:2' Estado = 22; *)
                Estado := 22;
            END_IF;


            IF temp10 THEN 
                is_DRIVE := UPMRacing_14E_StateMachine_IN_Accelerate;
                (* Entry 'Accelerate': '<S1>:146' *)
                (* '<S1>:146:2' Estado = 21; *)
                Estado := 21;
            END_IF;

            (* During 'ERROR_INVERTER': '<S1>:381' *)
            (* '<S1>:381:2' [Inverter_Error,Inverter_Warning] = Error_Control(AMK_bError1,AMK_bError2,AMK_bError3,AMK_bError4,AMK_bWarn1,AMK_bWarn2,AMK_bWarn3,AMK_bWarn4); *)
            (* Simulink Function 'Error_Control': '<S1>:390' *)
            b_AMK_bError1 := AMK_bError1;
            b_AMK_bError2 := AMK_bError2;
            b_AMK_bError3 := AMK_bError3;
            b_AMK_bError4 := AMK_bError4;
            b_AMK_bWarn1 := AMK_bWarn1;
            b_AMK_bWarn2 := AMK_bWarn2;
            b_AMK_bWarn3 := AMK_bWarn3;
            b_AMK_bWarn4 := AMK_bWarn4;
            i0_Error_Control(ssMethodType := SS_OUTPUT, AMK_bError1 := b_AMK_bError1, AMK_bError2 := b_AMK_bError2, AMK_bError3 := b_AMK_bError3, AMK_bError4 := b_AMK_bError4, AMK_bWarn1 := b_AMK_bWarn1, AMK_bWarn2 := b_AMK_bWarn2, AMK_bWarn3 := b_AMK_bWarn3, AMK_bWarn4 := b_AMK_bWarn4);
            sf_internal_predicateOutput := i0_Error_Control.Inverter_Error;
            temp10 := i0_Error_Control.Inverter_Warning;
            LogicalOperator1 := temp10;
            LogicalOperator := sf_internal_predicateOutput;
            Inverter_Error := LogicalOperator;
            Inverter_Warning := LogicalOperator1;

            CASE is_ERROR_INVERTER OF
                UPMRacing_14E_StateMachine_IN_ERROR: 
                    (* Outport: '<Root>/Estado_Error' *)
                    Estado_Error := 12;
                    (* During 'ERROR': '<S1>:385' *)
                    (* '<S1>:388:1' sf_internal_predicateOutput = Inverter_Error == 0; *)

                    IF  NOT LogicalOperator THEN 
                        (* Transition: '<S1>:388' *)
                        is_ERROR_INVERTER := UPMRacing_14E_StateMachine_IN_NO_ERROR;
                        (* Outport: '<Root>/Estado_Error' *)
                        (* Entry 'NO_ERROR': '<S1>:384' *)
                        (* No hay errores *)
                        (* '<S1>:384:3' Estado_Error = 11; *)
                        Estado_Error := 11;
                    ELSE 
                        (* '<S1>:435:1' sf_internal_predicateOutput = Reset_Button > 3000; *)

                        IF Reset_Button > 3000 THEN 
                            (* Transition: '<S1>:435' *)
                            is_ERROR_INVERTER := UPMRacing_14E_StateMachine_IN_RESET_ERROR;
                            (* Outport: '<Root>/Estado_Error' *)
                            (* Entry 'RESET_ERROR': '<S1>:403' *)
                            (* Reseteamos errores *)
                            (* '<S1>:403:3' Estado_Error = 13; *)
                            Estado_Error := 13;
                        ELSE 
                            (* Hay errores *)
                            (* Esperar a boton de reset para resetear errores *)
                            (* '<S1>:385:6' Info_Inverter_Error = Error_Info(AMK_ErrorInfo1,AMK_ErrorInfo2,AMK_ErrorInfo3,AMK_ErrorInfo4,... *)
                            (* '<S1>:385:7'     AMK_bError1,AMK_bError2,AMK_bError3,AMK_bError4) *)
                            (* Simulink Function 'Error_Info': '<S1>:463' *)
                            b_AMK_ErrorInfo1 := AMK_ErrorInfo1;
                            b_AMK_ErrorInfo2 := AMK_ErrorInfo2;
                            b_AMK_ErrorInfo3 := AMK_ErrorInfo3;
                            b_AMK_ErrorInfo4 := AMK_ErrorInfo4;
                            AMK_bError1_b := AMK_bError1;
                            AMK_bError2_h := AMK_bError2;
                            AMK_bError3_d := AMK_bError3;
                            AMK_bError4_a := AMK_bError4;
                            i0_Error_Info(ssMethodType := SS_OUTPUT, AMK_ErrorInfo1 := b_AMK_ErrorInfo1, AMK_ErrorInfo2 := b_AMK_ErrorInfo2, AMK_ErrorInfo3 := b_AMK_ErrorInfo3, AMK_ErrorInfo4 := b_AMK_ErrorInfo4, AMK_bError1 := AMK_bError1_b, AMK_bError2 := AMK_bError2_h, AMK_bError3 := AMK_bError3_d, AMK_bError4 := AMK_bError4_a);
                            temp7 := i0_Error_Info.Info_Inverter_Error;
                            b_Add := temp7;
                            Info_Inverter_Error := b_Add;
                        END_IF;

                    END_IF;

                UPMRacing_14E_StateMachine_IN_NO_ERROR: 
                    (* Outport: '<Root>/Estado_Error' *)
                    Estado_Error := 11;
                    (* During 'NO_ERROR': '<S1>:384' *)
                    (* '<S1>:386:1' sf_internal_predicateOutput = Inverter_Error==1 &amp; Reset_Button == 0; *)

                    IF LogicalOperator AND (Reset_Button = 0) THEN 
                        (* Transition: '<S1>:386' *)
                        is_ERROR_INVERTER := UPMRacing_14E_StateMachine_IN_ERROR;
                        (* Outport: '<Root>/Estado_Error' *)
                        (* Entry 'ERROR': '<S1>:385' *)
                        (* Hay errores *)
                        (* Esperar a boton de reset para resetear errores *)
                        (* '<S1>:385:4' Estado_Error = 12; *)
                        Estado_Error := 12;
                    END_IF;

                ELSE
                    (* Outport: '<Root>/Estado_Error' *)
                    Estado_Error := 13;
                    (* During 'RESET_ERROR': '<S1>:403' *)
                    (* '<S1>:436:1' sf_internal_predicateOutput = Reset_Button < 300; *)

                    IF Reset_Button < 300 THEN 
                        (* Transition: '<S1>:436' *)
                        (* Exit 'RESET_ERROR': '<S1>:403' *)
                        (* '<S1>:403:6' Info_Inverter_Error = 0; *)
                        Info_Inverter_Error := 0;
                        is_ERROR_INVERTER := UPMRacing_14E_StateMachine_IN_NO_ERROR;
                        (* Outport: '<Root>/Estado_Error' incorporates:
                         *  Outport: '<Root>/Info_Inverter_Error' *)
                        (* Entry 'NO_ERROR': '<S1>:384' *)
                        (* No hay errores *)
                        (* '<S1>:384:3' Estado_Error = 11; *)
                        Estado_Error := 11;
                    ELSE 
                        (* Reseteamos errores *)
                        (* '<S1>:403:5' [AMK_bErrorReset1,AMK_bErrorReset2,AMK_bErrorReset3,AMK_bErrorReset4] = Error_RESET *)
                        (* Simulink Function 'Error_RESET': '<S1>:414' *)
                        i0_Error_RESET(ssMethodType := SS_OUTPUT);
                        sf_internal_predicateOutput := i0_Error_RESET.AMK_bErrorReset1;
                        temp10 := i0_Error_RESET.AMK_bErrorReset2;
                        temp8 := i0_Error_RESET.AMK_bErrorReset3;
                        temp9 := i0_Error_RESET.AMK_bErrorReset4;
                        OutportBufferForAMK_bErrorReset4 := temp9;
                        OutportBufferForAMK_bErrorReset3 := temp8;
                        OutportBufferForAMK_bErrorReset2 := temp10;
                        Compare := sf_internal_predicateOutput;
                        AMK_bErrorReset1 := Compare;
                        AMK_bErrorReset2 := OutportBufferForAMK_bErrorReset2;
                        AMK_bErrorReset3 := OutportBufferForAMK_bErrorReset3;
                        AMK_bErrorReset4 := OutportBufferForAMK_bErrorReset4;
                    END_IF;

            END_CASE;

            (* During 'BRAKE_LIGHT': '<S1>:519' *)

            CASE is_BRAKE_LIGHT OF
                UPMRacing_14E_StateMachine_IN_LIGHT_OFF: 
                    (* During 'LIGHT_OFF': '<S1>:520' *)
                    (* '<S1>:523:1' sf_internal_predicateOutput = Brake_Pedal <= Braking_OffSet; *)

                    IF Brake_Pedal <= Braking_OffSet THEN 
                        (* Transition: '<S1>:523' *)
                        is_BRAKE_LIGHT := UPMRacing_14E_StateMachine_IN_LIGHT_ON;
                        (* Entry 'LIGHT_ON': '<S1>:522' *)
                    ELSE 
                        (* '<S1>:520:3' Brake_Light = false; *)
                        Brake_Light := FALSE;
                    END_IF;

                ELSE
                    (* During 'LIGHT_ON': '<S1>:522' *)
                    (* '<S1>:524:1' sf_internal_predicateOutput = Brake_Pedal > Braking_OffSet; *)

                    IF Brake_Pedal > Braking_OffSet THEN 
                        (* Transition: '<S1>:524' *)
                        is_BRAKE_LIGHT := UPMRacing_14E_StateMachine_IN_LIGHT_OFF;
                        (* Entry 'LIGHT_OFF': '<S1>:520' *)
                    ELSE 
                        (* '<S1>:522:3' Brake_Light = true; *)
                        Brake_Light := TRUE;
                    END_IF;

            END_CASE;

            (* During 'COOLING_RIGHT': '<S1>:526' *)

            CASE is_COOLING_RIGHT OF
                UPMRacing_14E_StateMachine_IN_COOLING_OFF_RIGHT: 
                    (* During 'COOLING_OFF_RIGHT': '<S1>:612' *)
                    (* '<S1>:611:1' sf_internal_predicateOutput = Cooling_Enable == true; *)

                    IF Cooling_Enable THEN 
                        (* Transition: '<S1>:611' *)
                        (* Exit 'COOLING_OFF_RIGHT': '<S1>:612' *)
                        (* '<S1>:612:4' Cooling_Pumps_On = false; *)
                        Cooling_Pumps_On := FALSE;
                        is_COOLING_RIGHT := UPMRacing_14E_StateMachine_IN_FAN_OFF;
                        (* Entry 'FAN_OFF': '<S1>:527' *)
                    END_IF;

                UPMRacing_14E_StateMachine_IN_FAN_OFF: 
                    (* During 'FAN_OFF': '<S1>:527' *)
                    (* '<S1>:531:1' sf_internal_predicateOutput = (AMK_TempMotor1 > Motor_Upper_Temp) || ... *)
                    (* '<S1>:531:2' (AMK_TempMotor3 > Motor_Upper_Temp); *)

                    IF (AMK_TempMotor1 > Motor_Upper_Temp) OR (AMK_TempMotor3 > Motor_Upper_Temp) THEN 
                        (* Transition: '<S1>:531' *)
                        is_COOLING_RIGHT := UPMRacing_14E_StateMachine_IN_FAN_ON;
                        (* Entry 'FAN_ON': '<S1>:530' *)
                    ELSE 
                        (* '<S1>:609:1' sf_internal_predicateOutput = Cooling_Enable == false; *)

                        IF  NOT Cooling_Enable THEN 
                            (* Transition: '<S1>:609' *)
                            is_COOLING_RIGHT := UPMRacing_14E_StateMachine_IN_COOLING_OFF_RIGHT;
                            (* Entry 'COOLING_OFF_RIGHT': '<S1>:612' *)
                            (* '<S1>:612:2' Cooling_Pumps_On = false; *)
                            Cooling_Pumps_On := FALSE;
                            (* '<S1>:612:3' Fan_Left = false; *)
                            Fan_Left := FALSE;
                        ELSE 
                            (* '<S1>:527:2' Fan_Right = false; *)
                            Fan_Right := FALSE;
                        END_IF;

                    END_IF;

                UPMRacing_14E_StateMachine_IN_FAN_OFF_Speed: 
                    (* During 'FAN_OFF_Speed': '<S1>:533' *)
                    (* '<S1>:534:1' sf_internal_predicateOutput = Speed<Fan_Lower_Speed; *)

                    IF Speed < UINT_TO_REAL(Fan_Lower_Speed) THEN 
                        (* Transition: '<S1>:534' *)
                        is_COOLING_RIGHT := UPMRacing_14E_StateMachine_IN_FAN_ON;
                        (* Entry 'FAN_ON': '<S1>:530' *)
                    ELSE 
                        (* '<S1>:607:1' sf_internal_predicateOutput = Cooling_Enable == false; *)

                        IF  NOT Cooling_Enable THEN 
                            (* Transition: '<S1>:607' *)
                            is_COOLING_RIGHT := UPMRacing_14E_StateMachine_IN_COOLING_OFF_RIGHT;
                            (* Entry 'COOLING_OFF_RIGHT': '<S1>:612' *)
                            (* '<S1>:612:2' Cooling_Pumps_On = false; *)
                            Cooling_Pumps_On := FALSE;
                            (* '<S1>:612:3' Fan_Left = false; *)
                            Fan_Left := FALSE;
                        ELSE 
                            (* '<S1>:533:2' Fan_Right = false; *)
                            Fan_Right := FALSE;
                        END_IF;

                    END_IF;

                ELSE
                    (* During 'FAN_ON': '<S1>:530' *)
                    (* '<S1>:532:1' sf_internal_predicateOutput = (AMK_TempMotor1 < Motor_Lower_Temp) || ... *)
                    (* '<S1>:532:2' (AMK_TempMotor3 < Motor_Lower_Temp); *)

                    IF (AMK_TempMotor1 < Motor_Lower_Temp) OR (AMK_TempMotor3 < Motor_Lower_Temp) THEN 
                        (* Transition: '<S1>:532' *)
                        is_COOLING_RIGHT := UPMRacing_14E_StateMachine_IN_FAN_OFF;
                        (* Entry 'FAN_OFF': '<S1>:527' *)
                    ELSE 
                        (* '<S1>:608:1' sf_internal_predicateOutput = Cooling_Enable == false; *)

                        IF  NOT Cooling_Enable THEN 
                            (* Transition: '<S1>:608' *)
                            is_COOLING_RIGHT := UPMRacing_14E_StateMachine_IN_COOLING_OFF_RIGHT;
                            (* Entry 'COOLING_OFF_RIGHT': '<S1>:612' *)
                            (* '<S1>:612:2' Cooling_Pumps_On = false; *)
                            Cooling_Pumps_On := FALSE;
                            (* '<S1>:612:3' Fan_Left = false; *)
                            Fan_Left := FALSE;
                        ELSE 
                            (* '<S1>:535:1' sf_internal_predicateOutput = Speed>Fan_Upper_Speed; *)

                            IF Speed > UINT_TO_REAL(Fan_Upper_Speed) THEN 
                                (* Transition: '<S1>:535' *)
                                is_COOLING_RIGHT := UPMRacing_14E_StateMachine_IN_FAN_OFF_Speed;
                                (* Entry 'FAN_OFF_Speed': '<S1>:533' *)
                            ELSE 
                                (* '<S1>:530:2' Fan_Right = false; *)
                                Fan_Right := FALSE;
                            END_IF;

                        END_IF;

                    END_IF;

            END_CASE;

            (* During 'COOLING_LEFT': '<S1>:543' *)
            (* '<S1>:543:3' [AIM_TempInverter1,AIM_TempInverter2,AIM_TempInverter3,AIM_TempInverter4] = Temp_Inverter(AMK_TempInverter1,AMK_TempInverter2,AMK_TempInverter3,AMK_TempInverter4); *)
            (* Simulink Function 'Temp_Inverter': '<S1>:577' *)
            b_AMK_TempInverter1 := AMK_TempInverter1;
            b_AMK_TempInverter2 := AMK_TempInverter2;
            b_AMK_TempInverter3 := AMK_TempInverter3;
            b_AMK_TempInverter4 := AMK_TempInverter4;
            i0_Temp_Inverter(ssMethodType := SS_OUTPUT, AMK_TempInverter1 := b_AMK_TempInverter1, AMK_TempInverter2 := b_AMK_TempInverter2, AMK_TempInverter3 := b_AMK_TempInverter3, AMK_TempInverter4 := b_AMK_TempInverter4);
            temp3 := i0_Temp_Inverter.AIM_TempInverter1;
            temp4 := i0_Temp_Inverter.AIM_TempInverter2;
            temp5 := i0_Temp_Inverter.AIM_TempInverter3;
            temp6 := i0_Temp_Inverter.AIM_TempInverter4;
            DataTypeConversion3_e := temp6;
            DataTypeConversion1_c := temp5;
            DataTypeConversion2_f := temp4;
            DataTypeConversion_h := temp3;
            AIM_TempInverter1 := DataTypeConversion_h;
            AIM_TempInverter2 := DataTypeConversion2_f;
            AIM_TempInverter3 := DataTypeConversion1_c;
            AIM_TempInverter4 := DataTypeConversion3_e;
            (* '<S1>:543:4' [AIM_TempMotor1,AIM_TempMotor2,AIM_TempMotor3,AIM_TempMotor4] = Temp_Motor(AMK_TempMotor1,AMK_TempMotor2,AMK_TempMotor3,AMK_TempMotor4); *)
            (* Simulink Function 'Temp_Motor': '<S1>:593' *)
            b_AMK_TempMotor1 := AMK_TempMotor1;
            b_AMK_TempMotor2 := AMK_TempMotor2;
            b_AMK_TempMotor3 := AMK_TempMotor3;
            b_AMK_TempMotor4 := AMK_TempMotor4;
            i0_Temp_Motor(ssMethodType := SS_OUTPUT, AMK_TempMotor1 := b_AMK_TempMotor1, AMK_TempMotor2 := b_AMK_TempMotor2, AMK_TempMotor3 := b_AMK_TempMotor3, AMK_TempMotor4 := b_AMK_TempMotor4);
            temp3 := i0_Temp_Motor.AIM_TempMotor1;
            temp4 := i0_Temp_Motor.AIM_TempMotor2;
            temp5 := i0_Temp_Motor.AIM_TempMotor3;
            temp6 := i0_Temp_Motor.AIM_TempMotor4;
            DataTypeConversion3_p := temp6;
            DataTypeConversion1_g := temp5;
            DataTypeConversion2_e := temp4;
            DataTypeConversion_e := temp3;
            AIM_TempMotor1 := DataTypeConversion_e;
            AIM_TempMotor2 := DataTypeConversion2_e;
            AIM_TempMotor3 := DataTypeConversion1_g;
            AIM_TempMotor4 := DataTypeConversion3_p;
            (* '<S1>:543:5' [AIM_TempIGBT1,AIM_TempIGBT2,AIM_TempIGBT3,AIM_TempIGBT4] = Temp_IGBT(AMK_TempIGBT1,AMK_TempIGBT2,AMK_TempIGBT3,AMK_TempIGBT4); *)
            (* Simulink Function 'Temp_IGBT': '<S1>:644' *)
            b_AMK_TempIGBT1 := AMK_TempIGBT1;
            b_AMK_TempIGBT2 := AMK_TempIGBT2;
            b_AMK_TempIGBT3 := AMK_TempIGBT3;
            b_AMK_TempIGBT4 := AMK_TempIGBT4;
            i0_Temp_IGBT(ssMethodType := SS_OUTPUT, AMK_TempIGBT1 := b_AMK_TempIGBT1, AMK_TempIGBT2 := b_AMK_TempIGBT2, AMK_TempIGBT3 := b_AMK_TempIGBT3, AMK_TempIGBT4 := b_AMK_TempIGBT4);
            temp3 := i0_Temp_IGBT.AIM_TempIGBT1;
            temp4 := i0_Temp_IGBT.AIM_TempIGBT2;
            temp5 := i0_Temp_IGBT.AIM_TempIGBT3;
            temp6 := i0_Temp_IGBT.AIM_TempIGBT4;
            DataTypeConversion3_o := temp6;
            DataTypeConversion1_n := temp5;
            DataTypeConversion2_m := temp4;
            DataTypeConversion_b := temp3;
            AIM_TempIGBT1 := DataTypeConversion_b;
            AIM_TempIGBT2 := DataTypeConversion2_m;
            AIM_TempIGBT3 := DataTypeConversion1_n;
            AIM_TempIGBT4 := DataTypeConversion3_o;
            (* '<S1>:543:6' [AIM_bDerating1,AIM_bDerating2,AIM_bDerating3,AIM_bDerating4] = Derating(AMK_bDerating1,AMK_bDerating2,AMK_bDerating3,AMK_bDerating4); *)
            (* Simulink Function 'Derating': '<S1>:711' *)
            b_AMK_bDerating1 := AMK_bDerating1;
            b_AMK_bDerating2 := AMK_bDerating2;
            b_AMK_bDerating3 := AMK_bDerating3;
            b_AMK_bDerating4 := AMK_bDerating4;
            i0_Derating(ssMethodType := SS_OUTPUT, AMK_bDerating1 := b_AMK_bDerating1, AMK_bDerating2 := b_AMK_bDerating2, AMK_bDerating3 := b_AMK_bDerating3, AMK_bDerating4 := b_AMK_bDerating4);
            sf_internal_predicateOutput := i0_Derating.AIM_bDerating1;
            temp10 := i0_Derating.AIM_bDerating2;
            temp8 := i0_Derating.AIM_bDerating3;
            temp9 := i0_Derating.AIM_bDerating4;
            AMK_bDerating4_p := temp9;
            AMK_bDerating3_g := temp8;
            AMK_bDerating2_p := temp10;
            AMK_bDerating1_h := sf_internal_predicateOutput;
            AIM_bDerating1 := AMK_bDerating1_h;
            AIM_bDerating2 := AMK_bDerating2_p;
            AIM_bDerating3 := AMK_bDerating3_g;
            AIM_bDerating4 := AMK_bDerating4_p;
            (* '<S1>:543:7' [AIM_TorqueCurrent1,AIM_TorqueCurrent2,AIM_TorqueCurrent3,AIM_TorqueCurrent4] = TorqueCurrent(AMK_TorqueCurrent1,AMK_TorqueCurrent2,AMK_TorqueCurrent3,AMK_TorqueCurrent4); *)
            (* Simulink Function 'TorqueCurrent': '<S1>:675' *)
            b_AMK_TorqueCurrent1 := AMK_TorqueCurrent1;
            b_AMK_TorqueCurrent2 := AMK_TorqueCurrent2;
            b_AMK_TorqueCurrent3 := AMK_TorqueCurrent3;
            b_AMK_TorqueCurrent4 := AMK_TorqueCurrent4;
            i0_TorqueCurrent(ssMethodType := SS_OUTPUT, AMK_TorqueCurrent1 := b_AMK_TorqueCurrent1, AMK_TorqueCurrent2 := b_AMK_TorqueCurrent2, AMK_TorqueCurrent3 := b_AMK_TorqueCurrent3, AMK_TorqueCurrent4 := b_AMK_TorqueCurrent4);
            temp12 := i0_TorqueCurrent.AIM_TorqueCurrent1;
            temp13 := i0_TorqueCurrent.AIM_TorqueCurrent2;
            temp14 := i0_TorqueCurrent.AIM_TorqueCurrent3;
            temp15 := i0_TorqueCurrent.AIM_TorqueCurrent4;
            AMK_TorqueCurrent4_b := temp15;
            AMK_TorqueCurrent3_p := temp14;
            AMK_TorqueCurrent2_b := temp13;
            AMK_TorqueCurrent1_m := temp12;
            AIM_TorqueCurrent1 := AMK_TorqueCurrent1_m;
            AIM_TorqueCurrent2 := AMK_TorqueCurrent2_b;
            AIM_TorqueCurrent3 := AMK_TorqueCurrent3_p;
            AIM_TorqueCurrent4 := AMK_TorqueCurrent4_b;
            (* '<S1>:543:8' [AIM_TargetVelocity1,AIM_TargetVelocity2,AIM_TargetVelocity3,AIM_TargetVelocity4] = TargetVelocity(AMK_TargetVelocity1,AMK_TargetVelocity2,AMK_TargetVelocity3,AMK_TargetVelocity4); *)
            (* Simulink Function 'TargetVelocity': '<S1>:691' *)
            AMK_TargetVelocity1_g := AMK_TargetVelocity1;
            AMK_TargetVelocity2_m := AMK_TargetVelocity2;
            AMK_TargetVelocity3_m := AMK_TargetVelocity3;
            AMK_TargetVelocity4_b := AMK_TargetVelocity4;
            i0_TargetVelocity(ssMethodType := SS_OUTPUT, AMK_TargetVelocity1 := AMK_TargetVelocity1_g, AMK_TargetVelocity2 := AMK_TargetVelocity2_m, AMK_TargetVelocity3 := AMK_TargetVelocity3_m, AMK_TargetVelocity4 := AMK_TargetVelocity4_b);
            temp12 := i0_TargetVelocity.AIM_TargetVelocity1;
            temp13 := i0_TargetVelocity.AIM_TargetVelocity2;
            temp14 := i0_TargetVelocity.AIM_TargetVelocity3;
            temp15 := i0_TargetVelocity.AIM_TargetVelocity4;
            AMK_TargetVelocity4_p := temp15;
            AMK_TargetVelocity3_h := temp14;
            AMK_TargetVelocity2_c := temp13;
            AMK_TargetVelocity1_gb := temp12;
            AIM_TargetVelocity1 := AMK_TargetVelocity1_gb;
            AIM_TargetVelocity2 := AMK_TargetVelocity2_c;
            AIM_TargetVelocity3 := AMK_TargetVelocity3_h;
            AIM_TargetVelocity4 := AMK_TargetVelocity4_p;
            (* '<S1>:543:9' [AIM_TorqueLimitPositiv1,AIM_TorqueLimitPositiv2,AIM_TorqueLimitPositiv3,AIM_TorqueLimitPositiv4] = TorqueLimitPositiv(AMK_TorqueLimitPositiv1,AMK_TorqueLimitPositiv2,AMK_TorqueLimitPositiv3,AMK_TorqueLimitPositiv4); *)
            (* Simulink Function 'TorqueLimitPositiv': '<S1>:730' *)
            AMK_TorqueLimitPositiv1_c := AMK_TorqueLimitPositiv1;
            AMK_TorqueLimitPositiv2_l := AMK_TorqueLimitPositiv2;
            AMK_TorqueLimitPositiv3_i := AMK_TorqueLimitPositiv3;
            AMK_TorqueLimitPositiv4_h := AMK_TorqueLimitPositiv4;
            i0_TorqueLimitPositiv(ssMethodType := SS_OUTPUT, AMK_TorqueLimitPositiv1 := AMK_TorqueLimitPositiv1_c, AMK_TorqueLimitPositiv2 := AMK_TorqueLimitPositiv2_l, AMK_TorqueLimitPositiv3 := AMK_TorqueLimitPositiv3_i, AMK_TorqueLimitPositiv4 := AMK_TorqueLimitPositiv4_h);
            temp12 := i0_TorqueLimitPositiv.AIM_TorqueLimitPositiv1;
            temp13 := i0_TorqueLimitPositiv.AIM_TorqueLimitPositiv2;
            temp14 := i0_TorqueLimitPositiv.AIM_TorqueLimitPositiv3;
            temp15 := i0_TorqueLimitPositiv.AIM_TorqueLimitPositiv4;
            AMK_TorqueLimitPositiv4_l := temp15;
            AMK_TorqueLimitPositiv3_m := temp14;
            AMK_TorqueLimitPositiv2_o := temp13;
            AMK_TorqueLimitPositiv1_e := temp12;
            AIM_TorqueLimitPositiv1 := AMK_TorqueLimitPositiv1_e;
            AIM_TorqueLimitPositiv2 := AMK_TorqueLimitPositiv2_o;
            AIM_TorqueLimitPositiv3 := AMK_TorqueLimitPositiv3_m;
            AIM_TorqueLimitPositiv4 := AMK_TorqueLimitPositiv4_l;
            (* '<S1>:543:10' [AIM_ActualVelocity1,AIM_ActualVelocity2,AIM_ActualVelocity3,AIM_ActualVelocity4] = ActualVelocity(AMK_ActualVelocity1,AMK_ActualVelocity2,AMK_ActualVelocity3,AMK_ActualVelocity4); *)
            (* Simulink Function 'ActualVelocity': '<S1>:749' *)
            AMK_ActualVelocity1_b := AMK_ActualVelocity1;
            AMK_ActualVelocity2_n := AMK_ActualVelocity2;
            AMK_ActualVelocity3_f := AMK_ActualVelocity3;
            AMK_ActualVelocity4_k := AMK_ActualVelocity4;
            i0_ActualVelocity(ssMethodType := SS_OUTPUT, AMK_ActualVelocity1 := AMK_ActualVelocity1_b, AMK_ActualVelocity2 := AMK_ActualVelocity2_n, AMK_ActualVelocity3 := AMK_ActualVelocity3_f, AMK_ActualVelocity4 := AMK_ActualVelocity4_k);
            temp12 := i0_ActualVelocity.AIM_ActualVelocity1;
            temp13 := i0_ActualVelocity.AIM_ActualVelocity2;
            temp14 := i0_ActualVelocity.AIM_ActualVelocity3;
            temp15 := i0_ActualVelocity.AIM_ActualVelocity4;
            AMK_ActualVelocity4_c := temp15;
            AMK_ActualVelocity3_i := temp14;
            AMK_ActualVelocity2_e := temp13;
            AMK_ActualVelocity1_l := temp12;
            AIM_ActualVelocity1 := AMK_ActualVelocity1_l;
            AIM_ActualVelocity2 := AMK_ActualVelocity2_e;
            AIM_ActualVelocity3 := AMK_ActualVelocity3_i;
            AIM_ActualVelocity4 := AMK_ActualVelocity4_c;
            (* '<S1>:543:11' [AIM_MagnetizingCurrent1,AIM_MagnetizingCurrent2,AIM_MagnetizingCurrent3,AIM_MagnetizingCurrent4] = MagnetizingCurrent(AMK_MagnetizingCurrent1,AMK_MagnetizingCurrent2,AMK_MagnetizingCurrent3,AMK_MagnetizingCurrent4); *)
            (* Simulink Function 'MagnetizingCurrent': '<S1>:653' *)
            b_AMK_MagnetizingCurrent1 := AMK_MagnetizingCurrent1;
            b_AMK_MagnetizingCurrent2 := AMK_MagnetizingCurrent2;
            b_AMK_MagnetizingCurrent3 := AMK_MagnetizingCurrent3;
            b_AMK_MagnetizingCurrent4 := AMK_MagnetizingCurrent4;
            i0_MagnetizingCurrent(ssMethodType := SS_OUTPUT, AMK_MagnetizingCurrent1 := b_AMK_MagnetizingCurrent1, AMK_MagnetizingCurrent2 := b_AMK_MagnetizingCurrent2, AMK_MagnetizingCurrent3 := b_AMK_MagnetizingCurrent3, AMK_MagnetizingCurrent4 := b_AMK_MagnetizingCurrent4);
            temp12 := i0_MagnetizingCurrent.AIM_MagnetizingCurrent1;
            temp13 := i0_MagnetizingCurrent.AIM_MagnetizingCurrent2;
            temp14 := i0_MagnetizingCurrent.AIM_MagnetizingCurrent3;
            temp15 := i0_MagnetizingCurrent.AIM_MagnetizingCurrent4;
            AMK_MagnetizingCurrent4_m := temp15;
            AMK_MagnetizingCurrent3_f := temp14;
            AMK_MagnetizingCurrent2_a := temp13;
            AMK_MagnetizingCurrent1_j := temp12;
            AIM_MagnetizingCurrent1 := AMK_MagnetizingCurrent1_j;
            AIM_MagnetizingCurrent2 := AMK_MagnetizingCurrent2_a;
            AIM_MagnetizingCurrent3 := AMK_MagnetizingCurrent3_f;
            AIM_MagnetizingCurrent4 := AMK_MagnetizingCurrent4_m;
            (* '<S1>:543:12' [AIM_ErrorInfo1,AIM_ErrorInfo2,AIM_ErrorInfo3,AIM_ErrorInfo4,AIM_bError1,AIM_bError2,AIM_bError3,AIM_bError4] = ErrorInfo(AMK_ErrorInfo1,AMK_ErrorInfo2,AMK_ErrorInfo3,AMK_ErrorInfo4,AMK_bError1,AMK_bError2,AMK_bError3,AMK_bError4) *)
            (* Simulink Function 'ErrorInfo': '<S1>:885' *)
            AMK_ErrorInfo1_n := AMK_ErrorInfo1;
            AMK_ErrorInfo2_f := AMK_ErrorInfo2;
            AMK_ErrorInfo3_l := AMK_ErrorInfo3;
            AMK_ErrorInfo4_o := AMK_ErrorInfo4;
            AMK_bError1_d := AMK_bError1;
            AMK_bError2_g := AMK_bError2;
            AMK_bError3_p := AMK_bError3;
            AMK_bError4_p := AMK_bError4;
            i0_ErrorInfo(ssMethodType := SS_OUTPUT, AMK_ErrorInfo1 := AMK_ErrorInfo1_n, AMK_ErrorInfo2 := AMK_ErrorInfo2_f, AMK_ErrorInfo3 := AMK_ErrorInfo3_l, AMK_ErrorInfo4 := AMK_ErrorInfo4_o, AMK_bError1 := AMK_bError1_d, AMK_bError2 := AMK_bError2_g, AMK_bError3 := AMK_bError3_p, AMK_bError4 := AMK_bError4_p);
            temp7 := i0_ErrorInfo.AIM_ErrorInfo1;
            tmp := i0_ErrorInfo.AIM_ErrorInfo2;
            temp1 := i0_ErrorInfo.AIM_ErrorInfo3;
            temp2 := i0_ErrorInfo.AIM_ErrorInfo4;
            sf_internal_predicateOutput := i0_ErrorInfo.AIM_bError1;
            temp10 := i0_ErrorInfo.AIM_bError2;
            temp8 := i0_ErrorInfo.AIM_bError3;
            temp9 := i0_ErrorInfo.AIM_bError4;
            AMK_bError4_g := temp9;
            AMK_bError3_n := temp8;
            AMK_bError2_e := temp10;
            AMK_bError1_k := sf_internal_predicateOutput;
            AMK_ErrorInfo4_oa := temp2;
            AMK_ErrorInfo3_p := temp1;
            AMK_ErrorInfo2_a := tmp;
            AMK_ErrorInfo1_h := temp7;
            AIM_ErrorInfo1 := AMK_ErrorInfo1_h;
            AIM_ErrorInfo2 := AMK_ErrorInfo2_a;
            AIM_ErrorInfo3 := AMK_ErrorInfo3_p;
            AIM_ErrorInfo4 := AMK_ErrorInfo4_oa;
            AIM_bError1 := AMK_bError1_k;
            AIM_bError2 := AMK_bError2_e;
            AIM_bError3 := AMK_bError3_n;
            AIM_bError4 := AMK_bError4_g;

